// TIA Portal V17 export
// export: Created 2024-08-09T12:53:15.349663Z, ExportSetting WithDefaults, DisplayName Totally Integrated Automation Portal, DisplayVersion V17 Update 7, DisplayName TIA Portal Openness, DisplayVersion V17 Update 7, DisplayName TIA Portal Version Control Interface, DisplayVersion V17, DisplayName STEP 7 Professional, DisplayVersion V17 Update 7, DisplayName STEP 7 Safety, DisplayVersion V17 Update 6, DisplayName WinCC Professional, DisplayVersion V17 Update 7
VAR_GLOBAL   // PLC tag table "Dec_Niveaux_DosCompo"
END_VAR
VAR_GLOBAL CONSTANT   // user constants
   NIV_DOSCOMPO_ATT_DEM_CIR : USInt := 10;
   NIV_DOSCOMPO_DEM_CIR : USInt := 20;
   NIV_DOSCOMPO_CHARG_EC : USInt := 40;
   NIV_DOSCOMPO_VID_CIR : USInt := 60;
   NIV_DOSCOMPO_VID_BEN : USInt := 80;
   NIV_DOSCOMPO_FVID_CIR : USInt := 160;
   NIV_DOSCOMPO_ATT_FINLOT : USInt := 200;
END_VAR
